(* IEC 61131-3 sources: volt/packages/volt-lsp-iec/test-corpus/bakon-nano/Device/Plc Logic/Application/Library Manager/(unresolved)/iecvaraccess3 interfaces, 57 files *)

(* ---- ACCESSRIGHTS.dut ---- *)
TYPE ACCESSRIGHTS :
(
	AR_NONE := 0,
	AR_READ := 1,
	AR_WRITE := 2,
	AR_READWRITE := 3,
	AR_EXECUTE := 8,
	AR_READEXECUTE := 9,
	AR_WRITEEXECUTE := 10,
	AR_READWRITEEXECUTE := 11
);
END_TYPE

(* ---- ARRAYDIMENSION.dut ---- *)
TYPE ARRAYDIMENSION :
STRUCT
	MINRANGE : DINT;
	MAXRANGE : DINT;
END_STRUCT
END_TYPE

(* ---- CONTENTFEATUREFLAGS.dut ---- *)
TYPE CONTENTFEATUREFLAGS :
(
	NONE := 16#0,
	SUPPORTOPCUA := 16#1,
	INCLUDECOMMENTS := 16#2,
	INCLUDEATTRIBUTES := 16#4,
	INCLUDETYPENODEATTRIBUTES := 16#8,
	INCLUDEEXECUTABLES := 16#10,
	USEEMPTYNAMESPACEBYDEFAULT := 16#20,
	OPCUAINFORMATIONMODEL := 16#40,
	OPCUACONTROLBROWSINGINIEC := 16#80,
	STRINGSASUTF8 := 16#100,
	USERMANAGEMENT := 16#200,
	CHECKINSTANCEACCESSRIGHTS := 16#400,
	CONTAINSALARMS := 16#800,
	NODEIDASSTRING := 16#1000
);
END_TYPE

(* ---- ENUMATTRIBUTES.dut ---- *)
TYPE ENUMATTRIBUTES :
STRUCT
	NNUMOFATTRIBUTES : WORD;
	PATTRIBUTES : POINTER TO ARRAY [0..0] OF POINTER TO STRING;
END_STRUCT
END_TYPE

(* ---- ENUMVALUES.dut ---- *)
TYPE ENUMVALUES :
STRUCT
	PVALUENAME : POINTER TO STRING;
	VALUE : LWORD;
END_STRUCT
END_TYPE

(* ---- HANDLESTORE.dut ---- *)
TYPE HANDLESTORE :
UNION
	HANDLE : RTS_IEC_HANDLE;
	DUMMY : ARRAY [0..1] OF DWORD;
END_UNION
END_TYPE

(* ---- IECVARACCSYMBOLSETDESCRIPTION.dut ---- *)
TYPE IECVARACCSYMBOLSETDESCRIPTION :
STRUCT
	PSZSYMBOLSSETNAME : POINTER TO STRING;
	DWSYMBOLSSETBIT : DWORD;
END_STRUCT
END_TYPE

(* ---- NAMESPACENODEFLAGS.dut ---- *)
TYPE NAMESPACENODEFLAGS :
(
	NONE := 0,
	NODETYPEMASK := 16#FF,
	NODETYPEBRANCHNODE := 16#1,
	NODETYPELEAFNODE := 16#2,
	BRANCHNODEINFOMASK := 16#FF00,
	BRANCHNODEIMPLICITROOTNODE := 16#100,
	BRANCHNODEAPPLICATIONNAME := 16#200,
	BRANCHNODELIBRARYNAMESPACE := 16#400,
	BRANCHNODEEXPLICITNAMESPACE := 16#800,
	BRANCHNODEMEMBERACCESS := 16#1000,
	SIGTYPENODEMASK := LWORD#4294901760,
	SIGTYPEGVL := 16#10000,
	SIGTYPEPROGRAM := 16#20000,
	SIGTYPEFB := 16#40000,
	SIGTYPESTRUCT := 16#80000,
	SIGTYPEMETHOD := 16#100000,
	SIGTYPEACTION := 16#200000,
	SIGTYPEPROPERTY := 16#400000,
	SIGTYPETRANSITION := 16#800000,
	SIGTYPEFUNCTION := 16#1000000,
	EXPORTEDVARIABLETYPEMASK := 16#FF00000000,
	EXPORTEDVARIABLEFLAG := 16#100000000,
	EXPORTEDSTATICVARIABLEFLAG := 16#200000000,
	EXPORTEDPROPERTYVARIABLEFLAG := 16#400000000,
	EXPORTEDVARIABLE := (ExportedVariableFlag + NodeTypeLeafNode),
	EXPORTEDSTATICVARIABLE := (ExportedStaticVariableFlag + NodeTypeLeafNode),
	EXPORTEDPROPERTYVARIABLE := (ExportedPropertyVariableFlag + NodeTypeLeafNode),
	NODEFLAGSMASK := 16#FF0000000000,
	NODEFLAGHIDDEN := 16#100000000000
);
END_TYPE

(* ---- RTSBROWSEINFO.dut ---- *)
TYPE RTSBROWSEINFO :
STRUCT
	HNODE : IBaseTreeNode;
	HTYPE : ITypeDesc;
	NARRAYINDEX : DINT;
	NSTRUCTINDEX : DINT;
END_STRUCT
END_TYPE

(* ---- TREENODETYPE.dut ---- *)
TYPE TREENODETYPE :
(
	BRANCHNODE := 4892,
	LEAFNODE := 1549,
	IECVARACCLEAFNODE := 8798,
	DATASERVERVARACCLEAFNODE := 1989
);
END_TYPE

(* ---- TYPEDESCARRAYASSTRUCT.dut ---- *)
TYPE TYPEDESCARRAYASSTRUCT :
STRUCT
	_DWSIZE : XWORD;
	_DWNATIVESIZE : XWORD;
	_IDIMENSIONS : INT;
	_DIMENSION : ARRAY [0..2] OF ArrayDimension;
	_PIBASETYPEDESC : ITypeDesc;
END_STRUCT
END_TYPE

(* ---- TYPEDESCASUNION.dut ---- *)
TYPE TYPEDESCASUNION :
STRUCT
	_TYPECLASS : TypeClass;
	_UNION : TypeDescUnion;
END_STRUCT
END_TYPE

(* ---- TYPEDESCSIMPLEASSTRUCT.dut ---- *)
TYPE TYPEDESCSIMPLEASSTRUCT :
STRUCT
	_DWSIZE : XWORD;
	_DWSWAPSIZE : XWORD;
END_STRUCT
END_TYPE

(* ---- TYPEDESCSTRUCTASSTRUCT.dut ---- *)
TYPE TYPEDESCSTRUCTASSTRUCT :
STRUCT
	_DWSIZE : XWORD;
	_DWNATIVESIZE : XWORD;
	_ICOMPONENTS : DINT;
	_COMPONENTS : POINTER TO ARRAY [0..0] OF IBaseTreeNode;
END_STRUCT
END_TYPE

(* ---- TYPEDESCUNION.dut ---- *)
TYPE TYPEDESCUNION :
UNION
	_SIMPLE : TypeDescSimpleAsStruct;
	_ARRAY : TypeDescArrayAsStruct;
	_STRUCT : TypeDescStructAsStruct;
END_UNION
END_TYPE

(* ---- TYPEDESCVARARRAYASSTRUCT.dut ---- *)
TYPE TYPEDESCVARARRAYASSTRUCT :
STRUCT
	_IDIMENSIONS : USINT;
	_DIMINFOOFFSET : __XWORD;
	_IDIMINFOTYPEDESC : ITypeDesc;
	_IBASETYPEDESC : ITypeDesc;
END_STRUCT
END_TYPE

(* ---- VARIABLEINFORMATIONSTRUCT.dut ---- *)
TYPE VARIABLEINFORMATIONSTRUCT :
STRUCT
	WSTRUCTSIZE : WORD;
	WFLAGS : WORD;
	DWOFFSET : XWORD;
	BYBITOFFSET : BYTE;
	XWMONITORINGOFFSET : XWORD;
END_STRUCT
END_TYPE

(* ---- VARIABLEINFORMATIONSTRUCT2.dut ---- *)
TYPE VARIABLEINFORMATIONSTRUCT2 :
STRUCT
	WSTRUCTSIZE : WORD;
	WFLAGS : WORD;
	DWOFFSET : XWORD;
	BYBITOFFSET : BYTE;
	XWMONITORINGOFFSET : XWORD;
	XWMONITORINGSIZE : XWORD;
END_STRUCT
END_TYPE

(* ---- VARIABLEINFORMATIONSTRUCT3.dut ---- *)
TYPE VARIABLEINFORMATIONSTRUCT3 :
STRUCT
	WSTRUCTSIZE : WORD;
	WFLAGS : WORD;
	DWOFFSET : XWORD;
	BYBITOFFSET : BYTE;
	XWMONITORINGOFFSET : XWORD;
	XWMONITORINGSIZE : XWORD;
	DWARRAYOFARRAYNESTING : DWORD;
	HBROWSEINFO : RTS_IEC_HANDLE;
	ABROWSEINFOPOOL : ARRAY [0..27] OF BYTE;
END_STRUCT
END_TYPE

(* ---- VARIABLEINFORMATIONSTRUCT4.dut ---- *)
TYPE VARIABLEINFORMATIONSTRUCT4 :
STRUCT
	WSTRUCTSIZE : WORD;
	WFLAGS : WORD;
	DWOFFSET : XWORD;
	BYBITOFFSET : BYTE;
	WMETHODMEMBERINDEX : WORD;
	XWMONITORINGOFFSET : XWORD;
	XWMONITORINGSIZE : XWORD;
	DWARRAYOFARRAYNESTING : DWORD;
	HBROWSEINFO : RTS_IEC_HANDLE;
	ABROWSEINFOPOOL : ARRAY [0..27] OF BYTE;
END_STRUCT
END_TYPE

(* ---- VARIABLEINFORMATIONSTRUCT5.dut ---- *)
TYPE VARIABLEINFORMATIONSTRUCT5 :
STRUCT
	WSTRUCTSIZE : WORD;
	WFLAGS : WORD;
	DWOFFSET : XWORD;
	BYBITOFFSET : BYTE;
	WMETHODMEMBERINDEX : WORD;
	XWMONITORINGOFFSET : XWORD;
	XWMONITORINGSIZE : XWORD;
	DWARRAYOFARRAYNESTING : DWORD;
	HBROWSEINFO : RTS_IEC_HANDLE;
	USER : HandleStore;
	VARINSTANCE : HandleStore;
	ARESERVED : ARRAY [0..11] OF BYTE;
END_STRUCT
END_TYPE

(* ---- VARIABLEINFORMATIONSTRUCT6.dut ---- *)
TYPE VARIABLEINFORMATIONSTRUCT6 :
STRUCT
	WSTRUCTSIZE : WORD;
	WFLAGS : WORD;
	DWOFFSET : XWORD;
	BYBITOFFSET : BYTE;
	WMETHODMEMBERINDEX : WORD;
	XWMONITORINGOFFSET : XWORD;
	XWMONITORINGSIZE : XWORD;
	DWARRAYOFARRAYNESTING : DWORD;
	HBROWSEINFO : RTS_IEC_HANDLE;
	USER : HandleStore;
	VARINSTANCE : HandleStore;
	CURRENTBROWSENAMEINDEX : DINT;
	ARESERVED : ARRAY [0..7] OF BYTE;
END_STRUCT
END_TYPE

(* ---- ARRAYDIMENSIONS.gvl ---- *)
VAR_GLOBAL
	MAX_ARRAY_DIMENSION : INT := 3;
END_VAR

(* ---- INTERFACEIDS.gvl ---- *)
VAR_GLOBAL
	ITFID_IIECVARACCESS3 : DWORD := 16#33;
	ITFID_IIECVARACCESS4 : DWORD := 16#48;
	ITFID_IIECVARACCESS5 : DWORD := 16#4F;
	ITFID_IIECVARACCESS6 : DWORD := 16#6B;
	ITFID_IIECVARACCESS7 : DWORD := 16#6C;
	ITFID_IIECVARACCESS8 : DWORD := 16#70;
	ITFID_IIECVARACCESS9 : DWORD := 16#72;
	ITFID_IIECVARACCESS10 : DWORD := 16#77;
	ITFID_IIECVARACCESS11 : DWORD := 16#79;
	ITFID_IIECVARACCESS12 : DWORD := 16#A0;
	ITFID_IIECVARACCESS13 : DWORD := 16#A4;
	ITFID_IIECVARACCESS14 : DWORD := 16#A5;
	ITFID_IIECVARACCESS15 : DWORD := 16#C8;
	ITFID_IIECVARACCESS16 : DWORD := 16#CA;
	ITFID_IIECVARACCESS17 : DWORD := 16#CF;
	ITFID_IIECVARACCESS18 : DWORD := 16#D0;
	ITFID_IVARIABLEINFORMATION : DWORD := 16#1001;
	ITFID_IGETTOPLEVELNODE : DWORD := 16#1002;
	ITFID_IVARIABLEINFORMATION2 : DWORD := 16#1003;
	ITFID_IVARIABLEINFORMATION3 : DWORD := 16#1104;
	ITFID_IVARIABLEINFORMATION4 : DWORD := 16#1106;
	ITFID_IVARIABLEINFORMATION5 : DWORD := 16#1107;
END_VAR

(* ---- NAMESPACENODEFLAGSEX.gvl ---- *)
VAR_GLOBAL
	NAMESPACENODEFLAGSEX_EXPORTEDEXECUTABLEVARIABLEFLAG : NamespaceNodeFlags := 16#800000000;
	NAMESPACENODEFLAGSEX_EXPORTEDEXECUTABLEVARIABLE : NamespaceNodeFlags := 16#800000002;
	NAMESPACENODEFLAGSEX_NODEHASEXECUTABLECHILDREN : NamespaceNodeFlags := 16#200000000000;
END_VAR

(* ---- TYPECLASSFLAGS.gvl ---- *)
VAR_GLOBAL
	TCF_GET_TYPE : DWORD := 0;
	TCF_GET_BASE_TYPE : DWORD := 1;
	TCF_GET_POU_TYPE : DWORD := 2;
	TCF_GET_ENUM_TYPE : DWORD := 4;
	TCF_GET_ALIAS_TYPE : DWORD := 8;
	TCF_GET_UA_BUILTIN_TYPE : DWORD := 16#10;
END_VAR

(* ---- VARIABLEINFORMATIONFLAGS.gvl ---- *)
VAR_GLOBAL
	VIF_COMPLETE_ACCESS : WORD := 16#1;
	VIF_DONT_MODIFY_OFFSET : WORD := 16#2;
	VIF_BITACCESS : WORD := 16#4;
	VIF_SPLIT_HUGE_VARIABLES : WORD := 16#8;
	VIF_CLIENT_ADDRESS_RESOLUTION : WORD := 16#10;
	VIF_NATIVE_SIZE : WORD := 16#20;
	VIF_EXTENDED_INFORMATION : WORD := 16#40;
	VIF_EXECUTABLE_MEMBER : WORD := 16#80;
END_VAR

(* ---- IIECVARACCESS10.itf ---- *)
INTERFACE IIECVARACCESS10
END_INTERFACE

METHOD VARACCGETNAMESPACENODEFLAGS : NamespaceNodeFlags
VAR_INPUT
	PNODE : IBaseTreeNode;
	PRESULT : POINTER TO UDINT;
END_VAR
END_METHOD

(* ---- IIECVARACCESS11.itf ---- *)
INTERFACE IIECVARACCESS11
END_INTERFACE

METHOD VARACCEXECUTECALL : RTS_IEC_RESULT
VAR_INPUT
	PNODE : IBaseTreeNode;
	PVARIABLEINFORMATION : POINTER TO VariableInformationStruct;
	PARGUMENTBUFFER : POINTER TO BYTE;
	NARGUMENTBUFFERSIZE : XWORD;
END_VAR
END_METHOD

METHOD VARACCGETENUMMEMBERATTRIBUTELIST : POINTER TO EnumAttributes
VAR_INPUT
	TYPEDESC : ITypeDesc;
	PNNUMOFENUMVALUES : POINTER TO INT;
	PRESULT : POINTER TO SysTypes.RTS_IEC_RESULT;
END_VAR
END_METHOD

METHOD VARACCGETNUMOFTYPEATTRIBUTES : WORD
VAR_INPUT
	TYPEDESC : ITypeDesc;
	PRESULT : POINTER TO SysTypes.RTS_IEC_RESULT;
END_VAR
END_METHOD

METHOD VARACCGETTYPEATTRIBUTEBYINDEX : POINTER TO STRING
VAR_INPUT
	TYPEDESC : ITypeDesc;
	WINDEX : WORD;
	PRESULT : POINTER TO SysTypes.RTS_IEC_RESULT;
END_VAR
END_METHOD

(* ---- IIECVARACCESS12.itf ---- *)
INTERFACE IIECVARACCESS12
END_INTERFACE

METHOD VARACCGETCONTENTFEATUREFLAGS : SysTypes.RTS_IEC_RESULT
VAR_INPUT
	PCONTENTFEATUREFLAGS : POINTER TO ContentFeatureFlags;
END_VAR
END_METHOD

METHOD VARACCGETRANGE : BOOL
VAR_INPUT
	TYPEDESC : ITypeDesc;
	PLOWER : POINTER TO LWORD;
	PUPPER : POINTER TO LWORD;
	PRESULT : POINTER TO SysTypes.RTS_IEC_RESULT;
END_VAR
END_METHOD

(* ---- IIECVARACCESS13.itf ---- *)
INTERFACE IIECVARACCESS13
END_INTERFACE

METHOD VARACCBROWSEDOWN3 : IBaseTreeNode
VAR_INPUT
	PNODE : ICollections.IBaseTreeNode;
	PVARIABLEINFORMATION : POINTER TO VariableInformationStruct2;
	BBROWSEINTOCOMPLEXTYPES : BOOL;
	PRESULT : POINTER TO SysTypes.RTS_IEC_RESULT;
END_VAR
END_METHOD

METHOD VARACCBROWSEGETCHILDBYINDEX2 : IBaseTreeNode
VAR_INPUT
	PNODE : IBaseTreeNode;
	DIINDEX : DINT;
	PVARIABLEINFORMATION : POINTER TO VariableInformationStruct2;
	PRESULT : POINTER TO UDINT;
END_VAR
END_METHOD

METHOD VARACCBROWSEGETNEXT3 : ICollections.IBaseTreeNode
VAR_INPUT
	PNODE : ICollections.IBaseTreeNode;
	PVARIABLEINFORMATION : POINTER TO VariableInformationStruct2;
	BBROWSEINTOCOMPLEXTYPES : BOOL;
	PRESULT : POINTER TO SysTypes.RTS_IEC_RESULT;
END_VAR
END_METHOD

METHOD VARACCBROWSEGETROOT2 : IBaseTreeNode
VAR_INPUT
	HUSER : RTS_IEC_HANDLE;
	PRESULT : POINTER TO UDINT;
END_VAR
END_METHOD

METHOD VARACCBROWSEUP3 : ICollections.IBaseTreeNode
VAR_INPUT
	PNODE : ICollections.IBaseTreeNode;
	PVARIABLEINFORMATION : POINTER TO VariableInformationStruct2;
	BBROWSEINTOCOMPLEXTYPES : BOOL;
	PRESULT : POINTER TO SysTypes.RTS_IEC_RESULT;
END_VAR
END_METHOD

METHOD VARACCGETACCESSRIGHTS2 : AccessRights
VAR_INPUT
	PNODE : IBaseTreeNode;
	PVARIABLEINFORMATION : POINTER TO VariableInformationStruct2;
	BGETUSERRIGHTS : BOOL;
	PRESULT : POINTER TO UDINT;
END_VAR
END_METHOD

METHOD VARACCGETAPPLICATIONNAME : RTS_IEC_RESULT
VAR_INPUT
	PSZAPPLICATIONNAME : POINTER TO STRING;
	NMAXLEN : DINT;
END_VAR
END_METHOD

METHOD VARACCINITVARINFO2 : SysTypes.RTS_IEC_RESULT
VAR_INPUT
	PVARIABLEINFORMATION : POINTER TO VariableInformationStruct2;
	NSIZEOFVARINFO : UINT;
	HUSER : RTS_IEC_HANDLE;
END_VAR
END_METHOD

(* ---- IIECVARACCESS14.itf ---- *)
INTERFACE IIECVARACCESS14
END_INTERFACE

METHOD VARACCGETREFERENCEBASETYPE : ITypeDesc
VAR_INPUT
	TYPEDESC : ITypeDesc;
	PRESULT : POINTER TO SysTypes.RTS_IEC_RESULT;
END_VAR
END_METHOD

(* ---- IIECVARACCESS15.itf ---- *)
INTERFACE IIECVARACCESS15
END_INTERFACE

METHOD VARACCGETTYPEDESCVARLENARRAY : RTS_IEC_RESULT
VAR_INPUT
	PTYPEDESC : ITypeDesc;
	PTYPEDESCSTRUCT : POINTER TO TypeDescVarArrayAsStruct;
END_VAR
END_METHOD

(* ---- IIECVARACCESS16.itf ---- *)
INTERFACE IIECVARACCESS16
END_INTERFACE

METHOD VARACCGETUABUILTINTYPE : USINT
VAR_INPUT
	TYPEDESC : ITypeDesc;
	PRESULT : POINTER TO RTS_IEC_RESULT;
END_VAR
END_METHOD

(* ---- IIECVARACCESS17.itf ---- *)
INTERFACE IIECVARACCESS17
END_INTERFACE

METHOD VARACCISREFERENCE : BOOL
VAR_INPUT
	PNODE : IBaseTreeNode;
	PVARIABLEINFORMATION : POINTER TO VariableInformationStruct;
	PRESULT : POINTER TO RTS_IEC_RESULT;
END_VAR
END_METHOD

(* ---- IIECVARACCESS18.itf ---- *)
INTERFACE IIECVARACCESS18
END_INTERFACE

METHOD VARACCFINDCHILDBYNAME : IBaseTreeNode
VAR_INPUT
	PNODE : IBaseTreeNode;
	PVARIABLEINFORMATION : POINTER TO VariableInformationStruct3;
	PNAME : POINTER TO STRING;
	PRESULT : POINTER TO RTS_IEC_RESULT;
END_VAR
END_METHOD

(* ---- IIECVARACCESS3.itf ---- *)
INTERFACE IIECVARACCESS3
END_INTERFACE

METHOD VARACCAPPENDVARIABLE : UDINT
VAR_INPUT
	PNODE : IBaseTreeNode;
END_VAR
END_METHOD

METHOD VARACCBEGINVARIABLECONFIGURATION : UDINT
VAR_INPUT
	BBLOCKING : BOOL;
END_VAR
END_METHOD

METHOD VARACCBROWSEDOWN : IBaseTreeNode
VAR_INPUT
	PNODE : IBaseTreeNode;
	PRESULT : POINTER TO UDINT;
END_VAR
END_METHOD

METHOD VARACCBROWSEGETNEXT : IBaseTreeNode
VAR_INPUT
	PNODE : IBaseTreeNode;
	PRESULT : POINTER TO UDINT;
END_VAR
END_METHOD

METHOD VARACCBROWSEGETROOT : IBaseTreeNode
VAR_INPUT
	PRESULT : POINTER TO UDINT;
END_VAR
END_METHOD

METHOD VARACCBROWSEUP : IBaseTreeNode
VAR_INPUT
	PNODE : IBaseTreeNode;
	PRESULT : POINTER TO UDINT;
END_VAR
END_METHOD

METHOD VARACCENDVARIABLECONFIGURATION : UDINT
END_METHOD

METHOD VARACCGETACCESSRIGHTS : AccessRights
VAR_INPUT
	PNODE : IBaseTreeNode;
	PRESULT : POINTER TO UDINT;
END_VAR
END_METHOD

METHOD VARACCGETADDRESS : POINTER TO BYTE
VAR_INPUT
	PNODE : IBaseTreeNode;
	PRESULT : POINTER TO UDINT;
END_VAR
END_METHOD

METHOD VARACCGETNODE : IBaseTreeNode
VAR_INPUT
	PSZPATH : POINTER TO STRING;
	PDWOFFSET : POINTER TO XWORD;
	PRESULT : POINTER TO UDINT;
END_VAR
END_METHOD

METHOD VARACCGETNODEFULLPATH : DINT
VAR_INPUT
	PNODE : IBaseTreeNode;
	PSZPATH : POINTER TO STRING;
	DIMAXPATH : DINT;
	PRESULT : POINTER TO UDINT;
END_VAR
END_METHOD

METHOD VARACCGETNODENAME : POINTER TO STRING
VAR_INPUT
	PNODE : IBaseTreeNode;
	PRESULT : POINTER TO UDINT;
END_VAR
END_METHOD

METHOD VARACCGETNODETYPE : TreeNodeType
VAR_INPUT
	PNODE : IBaseTreeNode;
	PRESULT : POINTER TO UDINT;
END_VAR
END_METHOD

METHOD VARACCGETSIZE : XWORD
VAR_INPUT
	PNODE : IBaseTreeNode;
	PRESULT : POINTER TO UDINT;
END_VAR
END_METHOD

METHOD VARACCGETSIZE2 : XWORD
VAR_INPUT
	PNODE : IBaseTreeNode;
	DWOFFSET : XWORD;
	PRESULT : POINTER TO UDINT;
END_VAR
END_METHOD

METHOD VARACCGETSWAPSIZE : XWORD
VAR_INPUT
	PNODE : IBaseTreeNode;
	PRESULT : POINTER TO UDINT;
END_VAR
END_METHOD

METHOD VARACCGETTYPECLASS : TypeClass
VAR_INPUT
	PNODE : IBaseTreeNode;
	PRESULT : POINTER TO UDINT;
END_VAR
END_METHOD

METHOD VARACCGETTYPEDESC : UDINT
VAR_INPUT
	PTYPEDESC : ITypeDesc;
	PTYPEDESCSTRUCT : POINTER TO TypeDescAsUnion;
END_VAR
END_METHOD

METHOD VARACCGETTYPENODE : ITypeDesc
VAR_INPUT
	PNODE : IBaseTreeNode;
	PRESULT : POINTER TO UDINT;
END_VAR
END_METHOD

METHOD VARACCGETVALUE : XWORD
VAR_INPUT
	PNODE : IBaseTreeNode;
	PDEST : POINTER TO BYTE;
	DWOFFSET : XWORD;
	DWSIZE : XWORD;
	PRESULT : POINTER TO UDINT;
END_VAR
END_METHOD

METHOD VARACCREMOVEVARIABLE : UDINT
VAR_INPUT
	PNODE : IBaseTreeNode;
END_VAR
END_METHOD

METHOD VARACCSETVALUE : XWORD
VAR_INPUT
	PNODE : IBaseTreeNode;
	PSRC : POINTER TO BYTE;
	DWOFFSET : XWORD;
	DWSIZE : XWORD;
	PRESULT : POINTER TO UDINT;
END_VAR
END_METHOD

METHOD VARACCSWAP : XWORD
VAR_INPUT
	PNODE : IBaseTreeNode;
	PDATA : POINTER TO BYTE;
	DWSIZE : XWORD;
	BMOTOROLA : BOOL;
	PRESULT : POINTER TO UDINT;
END_VAR
END_METHOD

METHOD VARACCSWAP2 : XWORD
VAR_INPUT
	PNODE : IBaseTreeNode;
	PDATA : POINTER TO BYTE;
	DWOFFSET : XWORD;
	BMOTOROLA : BOOL;
	PRESULT : POINTER TO UDINT;
END_VAR
END_METHOD

(* ---- IIECVARACCESS4.itf ---- *)
INTERFACE IIECVARACCESS4
END_INTERFACE

METHOD VARACCAPPENDVARIABLE : UDINT
VAR_INPUT
	PNODE : IBaseTreeNode;
END_VAR
END_METHOD

METHOD VARACCBEGINVARIABLECONFIGURATION : UDINT
VAR_INPUT
	BBLOCKING : BOOL;
END_VAR
END_METHOD

METHOD VARACCBROWSEDOWN : IBaseTreeNode
VAR_INPUT
	PNODE : IBaseTreeNode;
	PRESULT : POINTER TO UDINT;
END_VAR
END_METHOD

METHOD VARACCBROWSEGETNEXT : IBaseTreeNode
VAR_INPUT
	PNODE : IBaseTreeNode;
	PRESULT : POINTER TO UDINT;
END_VAR
END_METHOD

METHOD VARACCBROWSEGETROOT : IBaseTreeNode
VAR_INPUT
	PRESULT : POINTER TO UDINT;
END_VAR
END_METHOD

METHOD VARACCBROWSEUP : IBaseTreeNode
VAR_INPUT
	PNODE : IBaseTreeNode;
	PRESULT : POINTER TO UDINT;
END_VAR
END_METHOD

METHOD VARACCENDVARIABLECONFIGURATION : UDINT
END_METHOD

METHOD VARACCGETACCESSRIGHTS : AccessRights
VAR_INPUT
	PNODE : IBaseTreeNode;
	PRESULT : POINTER TO UDINT;
END_VAR
END_METHOD

METHOD VARACCGETADDRESS : POINTER TO BYTE
VAR_INPUT
	PNODE : IBaseTreeNode;
	PRESULT : POINTER TO UDINT;
END_VAR
END_METHOD

METHOD VARACCGETADDRESS2 : POINTER TO BYTE
VAR_INPUT
	PNODE : IBaseTreeNode;
	DWOFFSET : XWORD;
	PRESULT : POINTER TO UDINT;
END_VAR
END_METHOD

METHOD VARACCGETNODE : IBaseTreeNode
VAR_INPUT
	PSZPATH : POINTER TO STRING;
	PDWOFFSET : POINTER TO XWORD;
	PRESULT : POINTER TO UDINT;
END_VAR
END_METHOD

METHOD VARACCGETNODEFULLPATH : DINT
VAR_INPUT
	PNODE : IBaseTreeNode;
	PSZPATH : POINTER TO STRING;
	DIMAXPATH : DINT;
	PRESULT : POINTER TO UDINT;
END_VAR
END_METHOD

METHOD VARACCGETNODENAME : POINTER TO STRING
VAR_INPUT
	PNODE : IBaseTreeNode;
	PRESULT : POINTER TO UDINT;
END_VAR
END_METHOD

METHOD VARACCGETNODETYPE : TreeNodeType
VAR_INPUT
	PNODE : IBaseTreeNode;
	PRESULT : POINTER TO UDINT;
END_VAR
END_METHOD

METHOD VARACCGETSIZE : XWORD
VAR_INPUT
	PNODE : IBaseTreeNode;
	PRESULT : POINTER TO UDINT;
END_VAR
END_METHOD

METHOD VARACCGETSIZE2 : XWORD
VAR_INPUT
	PNODE : IBaseTreeNode;
	DWOFFSET : XWORD;
	PRESULT : POINTER TO UDINT;
END_VAR
END_METHOD

METHOD VARACCGETSWAPSIZE : XWORD
VAR_INPUT
	PNODE : IBaseTreeNode;
	PRESULT : POINTER TO UDINT;
END_VAR
END_METHOD

METHOD VARACCGETTYPECLASS : TypeClass
VAR_INPUT
	PNODE : IBaseTreeNode;
	PRESULT : POINTER TO UDINT;
END_VAR
END_METHOD

METHOD VARACCGETTYPEDESC : UDINT
VAR_INPUT
	PTYPEDESC : ITypeDesc;
	PTYPEDESCSTRUCT : POINTER TO TypeDescAsUnion;
END_VAR
END_METHOD

METHOD VARACCGETTYPENODE : ITypeDesc
VAR_INPUT
	PNODE : IBaseTreeNode;
	PRESULT : POINTER TO UDINT;
END_VAR
END_METHOD

METHOD VARACCGETTYPENODE2 : ITypeDesc
VAR_INPUT
	PNODE : IBaseTreeNode;
	DWOFFSET : XWORD;
	PRESULT : POINTER TO UDINT;
END_VAR
END_METHOD

METHOD VARACCGETVALUE : XWORD
VAR_INPUT
	PNODE : IBaseTreeNode;
	PDEST : POINTER TO BYTE;
	DWOFFSET : XWORD;
	DWSIZE : XWORD;
	PRESULT : POINTER TO UDINT;
END_VAR
END_METHOD

METHOD VARACCREMOVEVARIABLE : UDINT
VAR_INPUT
	PNODE : IBaseTreeNode;
END_VAR
END_METHOD

METHOD VARACCSETVALUE : XWORD
VAR_INPUT
	PNODE : IBaseTreeNode;
	PSRC : POINTER TO BYTE;
	DWOFFSET : XWORD;
	DWSIZE : XWORD;
	PRESULT : POINTER TO UDINT;
END_VAR
END_METHOD

METHOD VARACCSWAP : XWORD
VAR_INPUT
	PNODE : IBaseTreeNode;
	PDATA : POINTER TO BYTE;
	DWSIZE : XWORD;
	BMOTOROLA : BOOL;
	PRESULT : POINTER TO UDINT;
END_VAR
END_METHOD

METHOD VARACCSWAP2 : XWORD
VAR_INPUT
	PNODE : IBaseTreeNode;
	PDATA : POINTER TO BYTE;
	DWOFFSET : XWORD;
	BMOTOROLA : BOOL;
	PRESULT : POINTER TO UDINT;
END_VAR
END_METHOD

(* ---- IIECVARACCESS5.itf ---- *)
INTERFACE IIECVARACCESS5
END_INTERFACE

METHOD VARACCAPPENDVARIABLE3 : RTS_IEC_RESULT
VAR_INPUT
	PNODE : IBaseTreeNode;
	PVARIABLEINFORMATION : POINTER TO VariableInformationStruct;
END_VAR
END_METHOD

METHOD VARACCGETADDRESS3 : POINTER TO BYTE
VAR_INPUT
	PNODE : IBaseTreeNode;
	PVARIABLEINFORMATION : POINTER TO VariableInformationStruct;
	PRESULT : POINTER TO RTS_IEC_RESULT;
END_VAR
END_METHOD

METHOD VARACCGETNODE3 : IBaseTreeNode
VAR_INPUT
	PSZPATH : POINTER TO STRING;
	PVARIABLEINFORMATION : POINTER TO VariableInformationStruct;
	PRESULT : POINTER TO RTS_IEC_RESULT;
END_VAR
END_METHOD

METHOD VARACCGETNODEFULLPATH3 : DINT
VAR_INPUT
	PNODE : IBaseTreeNode;
	PVARIABLEINFORMATION : POINTER TO VariableInformationStruct;
	PSZPATH : POINTER TO STRING;
	DIMAXPATH : DINT;
	PRESULT : POINTER TO RTS_IEC_RESULT;
END_VAR
END_METHOD

METHOD VARACCGETNODENAME3 : POINTER TO STRING
VAR_INPUT
	PNODE : IBaseTreeNode;
	PVARIABLEINFORMATION : POINTER TO VariableInformationStruct;
	PRESULT : POINTER TO RTS_IEC_RESULT;
END_VAR
END_METHOD

METHOD VARACCGETSIZE3 : XWORD
VAR_INPUT
	PNODE : IBaseTreeNode;
	PVARIABLEINFORMATION : POINTER TO VariableInformationStruct;
	PRESULT : POINTER TO RTS_IEC_RESULT;
END_VAR
END_METHOD

METHOD VARACCGETTYPECLASS3 : TypeClass
VAR_INPUT
	PNODE : IBaseTreeNode;
	PVARIABLEINFORMATION : POINTER TO VariableInformationStruct;
	PRESULT : POINTER TO RTS_IEC_RESULT;
END_VAR
END_METHOD

METHOD VARACCGETTYPENODE3 : ITypeDesc
VAR_INPUT
	PNODE : IBaseTreeNode;
	PVARIABLEINFORMATION : POINTER TO VariableInformationStruct;
	PRESULT : POINTER TO RTS_IEC_RESULT;
END_VAR
END_METHOD

METHOD VARACCGETVALUE3 : XWORD
VAR_INPUT
	PNODE : IBaseTreeNode;
	PVARIABLEINFORMATION : POINTER TO VariableInformationStruct;
	PDEST : POINTER TO BYTE;
	DWSIZE : XWORD;
	PRESULT : POINTER TO RTS_IEC_RESULT;
END_VAR
END_METHOD

METHOD VARACCREMOVEVARIABLE3 : RTS_IEC_RESULT
VAR_INPUT
	PNODE : IBaseTreeNode;
	PVARIABLEINFORMATION : POINTER TO VariableInformationStruct;
END_VAR
END_METHOD

METHOD VARACCSETVALUE3 : XWORD
VAR_INPUT
	PNODE : IBaseTreeNode;
	PVARIABLEINFORMATION : POINTER TO VariableInformationStruct;
	PSRC : POINTER TO BYTE;
	DWSIZE : XWORD;
	PRESULT : POINTER TO RTS_IEC_RESULT;
END_VAR
END_METHOD

METHOD VARACCSWAP3 : XWORD
VAR_INPUT
	PNODE : IBaseTreeNode;
	PVARIABLEINFORMATION : POINTER TO VariableInformationStruct;
	PDATA : POINTER TO BYTE;
	BMOTOROLA : BOOL;
	PRESULT : POINTER TO RTS_IEC_RESULT;
END_VAR
END_METHOD

(* ---- IIECVARACCESS6.itf ---- *)
INTERFACE IIECVARACCESS6
END_INTERFACE

METHOD VARACCBROWSEGETCHILDBYINDEX : IBaseTreeNode
VAR_INPUT
	PNODE : IBaseTreeNode;
	DIINDEX : DINT;
	PRESULT : POINTER TO UDINT;
END_VAR
END_METHOD

(* ---- IIECVARACCESS7.itf ---- *)
INTERFACE IIECVARACCESS7
END_INTERFACE

METHOD VARACCENTERACCESS : SysTypes.RTS_IEC_RESULT
END_METHOD

METHOD VARACCGETATTRIBUTEBYINDEX : POINTER TO STRING
VAR_INPUT
	PNODE : IBaseTreeNode;
	WINDEX : WORD;
	PRESULT : POINTER TO SysTypes.RTS_IEC_RESULT;
END_VAR
END_METHOD

METHOD VARACCGETENUMVALUES : POINTER TO EnumValues
VAR_INPUT
	TYPEDESC : ITypeDesc;
	PNNUMOFENUMVALUES : POINTER TO INT;
	PRESULT : POINTER TO SysTypes.RTS_IEC_RESULT;
END_VAR
END_METHOD

METHOD VARACCGETNODEFLAGS : DWORD
VAR_INPUT
	PNODE : IBaseTreeNode;
	PRESULT : POINTER TO SysTypes.RTS_IEC_RESULT;
END_VAR
END_METHOD

METHOD VARACCGETNUMOFATTRIBUTES : WORD
VAR_INPUT
	PNODE : IBaseTreeNode;
	PRESULT : POINTER TO SysTypes.RTS_IEC_RESULT;
END_VAR
END_METHOD

METHOD VARACCGETNUMOFTYPES : DINT
VAR_INPUT
	PRESULT : POINTER TO RTS_IEC_RESULT;
END_VAR
END_METHOD

METHOD VARACCGETTYPECLASSFROMTYPE : TypeClass
VAR_INPUT
	TYPEDESC : ITypeDesc;
	DWFLAGS : DWORD;
	PRESULT : POINTER TO RTS_IEC_RESULT;
END_VAR
END_METHOD

METHOD VARACCGETTYPENAME : POINTER TO STRING
VAR_INPUT
	TYPEDESC : ITypeDesc;
	PRESULT : POINTER TO SysTypes.RTS_IEC_RESULT;
END_VAR
END_METHOD

METHOD VARACCGETTYPENODEBYINDEX : ITypeDesc
VAR_INPUT
	DIINDEX : DINT;
	PRESULT : POINTER TO RTS_IEC_RESULT;
END_VAR
END_METHOD

METHOD VARACCLEAVEACCESS : SysTypes.RTS_IEC_RESULT
END_METHOD

(* ---- IIECVARACCESS8.itf ---- *)
INTERFACE IIECVARACCESS8
END_INTERFACE

METHOD VARACCGETBASETYPE : ITypeDesc
VAR_INPUT
	TYPEDESC : ITypeDesc;
END_VAR
END_METHOD

METHOD VARACCHASBASETYPE : BOOL
VAR_INPUT
	TYPEDESC : ITypeDesc;
END_VAR
END_METHOD

(* ---- IIECVARACCESS9.itf ---- *)
INTERFACE IIECVARACCESS9
END_INTERFACE

METHOD VARACCBROWSEDOWN2 : IBaseTreeNode
VAR_INPUT
	PNODE : ICollections.IBaseTreeNode;
	PVARIABLEINFORMATION : POINTER TO VariableInformationStruct3;
	PRESULT : POINTER TO SysTypes.RTS_IEC_RESULT;
END_VAR
END_METHOD

METHOD VARACCBROWSEGETNEXT2 : ICollections.IBaseTreeNode
VAR_INPUT
	PNODE : ICollections.IBaseTreeNode;
	PVARIABLEINFORMATION : POINTER TO VariableInformationStruct3;
	PRESULT : POINTER TO SysTypes.RTS_IEC_RESULT;
END_VAR
END_METHOD

METHOD VARACCBROWSERECURSIVE : SysTypes.RTS_IEC_RESULT
VAR_INPUT
	PNODE : ICollections.IBaseTreeNode;
	PVARIABLEINFORMATION : POINTER TO VariableInformationStruct3;
	PFBROWSECALLBACK : POINTER TO BYTE;
	PUSERPARAMETER : POINTER TO BYTE;
END_VAR
END_METHOD

METHOD VARACCBROWSEUP2 : ICollections.IBaseTreeNode
VAR_INPUT
	PNODE : ICollections.IBaseTreeNode;
	PVARIABLEINFORMATION : POINTER TO VariableInformationStruct3;
	PRESULT : POINTER TO SysTypes.RTS_IEC_RESULT;
END_VAR
END_METHOD

METHOD VARACCEXITVARINFO : SysTypes.RTS_IEC_RESULT
VAR_INPUT
	PVARIABLEINFORMATION : POINTER TO VariableInformationStruct2;
END_VAR
END_METHOD

METHOD VARACCGETCLIENTOFFSET : XWORD
VAR_INPUT
	PNODE : IBaseTreeNode;
	PRESULT : POINTER TO SysTypes.RTS_IEC_RESULT;
END_VAR
END_METHOD

METHOD VARACCGETNODE4 : ICollections.IBaseTreeNode
VAR_INPUT
	PSZPATH : POINTER TO STRING;
	PVARIABLEINFORMATION : POINTER TO VariableInformationStruct3;
	PRESULT : POINTER TO SysTypes.RTS_IEC_RESULT;
END_VAR
END_METHOD

METHOD VARACCGETNODEFULLPATH4 : DINT
VAR_INPUT
	PNODE : ICollections.IBaseTreeNode;
	PVARIABLEINFORMATION : POINTER TO VariableInformationStruct3;
	PSZPATH : POINTER TO STRING;
	DIMAXPATH : DINT;
	PRESULT : POINTER TO SysTypes.RTS_IEC_RESULT;
END_VAR
END_METHOD

METHOD VARACCGETNODENAME4 : SysTypes.RTS_IEC_RESULT
VAR_INPUT
	PNODE : ICollections.IBaseTreeNode;
	PVARIABLEINFORMATION : POINTER TO VariableInformationStruct3;
	PSZNODENAME : POINTER TO STRING;
	NNODENAMELEN : UDINT;
END_VAR
END_METHOD

METHOD VARACCINITVARINFO : SysTypes.RTS_IEC_RESULT
VAR_INPUT
	PVARIABLEINFORMATION : POINTER TO VariableInformationStruct2;
	NSIZEOFVARINFO : UINT;
END_VAR
END_METHOD

(* ---- ITYPEDESC.itf ---- *)
INTERFACE ITYPEDESC
END_INTERFACE

METHOD FINDNODE : IInstancePathBuildingNode
VAR_INPUT
	PSTPATH : POINTER TO STRING;
	VARINFO : IVariableInformation;
	PRESULT : POINTER TO UDINT;
END_VAR
VAR_IN_OUT
	IOFFSETINPATH : DINT;
END_VAR
END_METHOD

METHOD GET : XWORD
VAR_INPUT
	PDEST : POINTER TO BYTE;
	PSRC : POINTER TO BYTE;
	VARINFO : IVariableInformation;
	DWSIZE : XWORD;
	PRESULT : POINTER TO UDINT;
END_VAR
END_METHOD

METHOD GETNATIVESIZE : XWORD
END_METHOD

METHOD GETSIZE : XWORD
END_METHOD

METHOD GETSIZE2 : XWORD
VAR_INPUT
	VARINFO : IVariableInformation;
END_VAR
END_METHOD

METHOD GETSWAPSIZE : XWORD
END_METHOD

METHOD GETTYPECLASS : TypeClass
END_METHOD

METHOD GETTYPEDESC : UDINT
VAR_INPUT
	PTYPEDESCSTRUCT : POINTER TO TypeDescAsUnion;
END_VAR
END_METHOD

METHOD GETTYPENODE : ITypeDesc
VAR_INPUT
	VARINFO : IVariableInformation;
END_VAR
END_METHOD

METHOD NODEFOUND : UDINT
VAR_INPUT
	VARINFO : IVariableInformation;
	BDIRECTCHILDFOUND : BOOL;
END_VAR
END_METHOD

METHOD SET : XWORD
VAR_INPUT
	PSRC : POINTER TO BYTE;
	PDEST : POINTER TO BYTE;
	VARINFO : IVariableInformation;
	DWSIZE : XWORD;
	PRESULT : POINTER TO UDINT;
END_VAR
END_METHOD

METHOD SWAP : XWORD
VAR_INPUT
	PDATA : POINTER TO BYTE;
	BMOTOROLA : BOOL;
	PRESULT : POINTER TO UDINT;
END_VAR
END_METHOD

METHOD SWAP2 : XWORD
VAR_INPUT
	PDATA : POINTER TO BYTE;
	VARINFO : IVariableInformation;
	BMOTOROLA : BOOL;
	PRESULT : POINTER TO UDINT;
END_VAR
END_METHOD

(* ---- ITYPEDESC2.itf ---- *)
INTERFACE ITYPEDESC2
END_INTERFACE

METHOD GETTYPECLASS2 : TypeClass
VAR_INPUT
	DWFLAGS : DWORD;
END_VAR
END_METHOD

(* ---- ITYPEDESC3.itf ---- *)
INTERFACE ITYPEDESC3
END_INTERFACE

METHOD GETENUMVALUES : POINTER TO EnumValues
VAR_INPUT
	PNNUMOFENUMVALUES : POINTER TO INT;
	PRESULT : POINTER TO RTS_IEC_RESULT;
END_VAR
END_METHOD

METHOD GETNAME : POINTER TO STRING
VAR_INPUT
	PRESULT : POINTER TO SysTypes.RTS_IEC_RESULT;
END_VAR
END_METHOD

(* ---- ITYPEDESC4.itf ---- *)
INTERFACE ITYPEDESC4
END_INTERFACE

METHOD GETNATIVESIZE2 : XWORD
VAR_INPUT
	VARINFO : IVariableInformation;
END_VAR
END_METHOD

(* ---- ITYPEDESCEXECUTABLE.itf ---- *)
INTERFACE ITYPEDESCEXECUTABLE
END_INTERFACE

METHOD GETDEFININGSIGNATURE : ITypeDesc4
END_METHOD

(* ---- ITYPEDESCSUBRANGE.itf ---- *)
INTERFACE ITYPEDESCSUBRANGE
END_INTERFACE

METHOD GETRANGE : BOOL
VAR_INPUT
	PLOWER : POINTER TO LWORD;
	PUPPER : POINTER TO LWORD;
END_VAR
END_METHOD

(* ---- ITYPEDESCWITHATTRIBUTES.itf ---- *)
INTERFACE ITYPEDESCWITHATTRIBUTES
END_INTERFACE

METHOD GETATTRIBUTEBYINDEX : POINTER TO STRING
VAR_INPUT
	WINDEX : WORD;
END_VAR
END_METHOD

METHOD GETENUMMEMBERATTRIBUTELIST : POINTER TO EnumAttributes
VAR_INPUT
	PNNUMOFENUMVALUES : POINTER TO INT;
	PRESULT : POINTER TO RTS_IEC_RESULT;
END_VAR
END_METHOD

METHOD GETNUMOFATTRIBUTES : WORD
END_METHOD

(* ---- ITYPEDESCWITHBASETYPE.itf ---- *)
INTERFACE ITYPEDESCWITHBASETYPE
END_INTERFACE

METHOD GETBASETYPE : ITypeDesc
END_METHOD

(* ---- ITYPEDESCWITHREFERENCETYPE.itf ---- *)
INTERFACE ITYPEDESCWITHREFERENCETYPE
END_INTERFACE

METHOD GETREFERENCEBASETYPE : ITypeDesc
END_METHOD

(* ---- IVARIABLEINFORMATION.itf ---- *)
INTERFACE IVARIABLEINFORMATION
END_INTERFACE

METHOD INCREMENTOFFSET : XWORD
VAR_INPUT
	DWTOINCREMENT : XWORD;
END_VAR
END_METHOD

(* ---- IVARIABLEINFORMATION2.itf ---- *)
INTERFACE IVARIABLEINFORMATION2
END_INTERFACE

(* ---- IVARIABLEINFORMATION3.itf ---- *)
INTERFACE IVARIABLEINFORMATION3
END_INTERFACE

(* ---- IVARIABLEINFORMATION4.itf ---- *)
INTERFACE IVARIABLEINFORMATION4
END_INTERFACE

(* ---- IVARIABLEINFORMATION5.itf ---- *)
INTERFACE IVARIABLEINFORMATION5
END_INTERFACE
